# EPICS substitutions: ipApp/iocsh/EXAMPLE_Pelco_CM6700.substitutions
file "$(IP)/ipApp/Db/Pelco_CM6700_names.db"
{
pattern
{STR}
{ZRST}
{ONST}
{TWST}
{THST}
{FRST}
{FVST}
{SXST}
{SVST}
{EIST}
{NIST}
{TEST}
{ELST}
{TVST}
{TTST}
{FTST}
{FFST}
}
